FUNCTION_BLOCK fbSliderWithGripperEM EXTENDS fbEM
VAR
	i : INT;
	state : INT;
	initial: BOOL := TRUE;
	servo_GO: BOOL;
	
	fbSignalSim: fbSignalSimSliderWithGripper;
END_VAR
VAR_INPUT
	
END_VAR
VAR_OUTPUT
	
END_VAR

(*
THIS fb use IOs listed below
DATA.I[1] -> true when gripper closed
DATA.I[2] -> true when gripper opened
DATA.I[3] -> part present
DATA.Q[1] -> 1 CLOSE / 0 OPEN gripper
DATA.Q[3] -> SERVO_GO
DATA.pick_pos -> desired pick position
DATA.drop_pos -> desired drop position
DATA.act_pos -> actual postition ( resolved in SIM or SERVO_HANDLER)
DATA.give_pos -> moves desired position into SIM or SERVO_HANDLER)
*)

GetUnCmd();
fbSignalSim(
	em := em,
	EnableSim := EnableSim,
	CmdSim := CmdSim
);

IF initial THEN // AFTER START OF PLC ENTER Undefined state
	state:=0;
	//em.CMD := E_CMD.powerOn; //// MAKES SENSE? <- no it doesnt because you change input 
	initial:= FALSE;
	 em.Config.Data.pick_pos:=10; 
	 em.Config.Data.pick_pos:=200;
	
END_IF

IF em.CMD = E_CMD.abort THEN
	state:=65;
END_IF

IF em.CMD = E_CMD.stop THEN
	state:=70;
END_IF

CASE state OF
	
	0:		//RESETTING
		em.Status := E_Status.resetting;	
		
		
		IF  em.Config.Data.pick_pos = em.Config.Data.act_pos THEN   // ACTUAL POS READ FROM SERVO HANDLER / FOR NOW FROM SIGNAL SIM
				
				servo_GO:=FALSE;
				state :=30; // IF gripper at PICK_pos go to idle
		END_IF
		IF em.CMD = E_CMD.reset THEN 		
				em.Config.Data.give_pos:=em.Config.Data.pick_pos;
				servo_GO:=TRUE;
				
				//// IF gripper pos unknown move to PICK
				//SERVO_HANDLER HAS TO KNOW THE CASE STEP TO DECIDE WHERE TO MOVE 			 
				//HERE SIGNAL SIM HANDLE THIS		
		END_IF
		

	
	30:		//IDLE
		em.Status := E_Status.idle;
		IF em.CMD = E_CMD.start THEN 
			state :=40;
		END_IF
		

	40:		//EXECUTE.1
		em.Status := E_Status.execute;
				
		//Close gripper when part present
		IF em.Config.Data.I[3]  THEN 
			em.Config.Data.Q[1]:= TRUE; //CLOSE GRIPPER
		END_IF
		
		//When Gripper closed --> state 41
		IF em.Config.Data.I[1] = TRUE AND em.Config.Data.I[2]=FALSE THEN
			state:=41;
		END_IF

	41:		//EXECUTE.2 ORDER TO MOVE TO CHOOSEN POSITION
		em.Status := E_Status.execute;
		em.Config.Data.give_pos := em.Config.Data.drop_pos;
		servo_GO:=TRUE; 							
		IF em.Config.Data.act_pos = em.Config.Data.drop_pos THEN
		servo_GO:=FALSE;
		state:=42;										
		END_IF


	42:		//EXECUTE.3 OPEN GRIPPER
	
		em.Status := E_Status.execute;
		em.Config.Data.Q[1]:=FALSE; //OPEN GRIPPER
		IF em.Config.Data.I[1] = FALSE AND em.Config.Data.I[2]=TRUE THEN
			state:=43;
		END_IF
		
			
	43:		//EXECUTE.4 MOVING PICK_POS WITHOUT PART

		em.Status := E_Status.execute;
		IF NOT em.Config.Data.I[3]  
			AND em.Config.Data.act_pos =em.Config.Data.drop_pos THEN//when part gone
			em.Config.Data.give_pos:=em.Config.Data.pick_pos;
			servo_GO:=TRUE;//GO 
			//SERVO_HANDLER HAS TO KNOW THE CASE STEP TO DECIDE WHERE TO MOVE 			 
			//HERE SIGNAL SIM HANDLE THIS	
		END_IF
		
		IF em.Config.Data.act_pos = em.Config.Data.pick_pos THEN
			servo_GO:=FALSE;
			state:=40;
			//em.Config.Data.pick_pos:= -1;
			//em.Config.Data.drop_pos:= -1;
		END_IF
	
	
	65:		//ABORTED

		em.Status := E_Status.aborted;	
		servo_GO:=FALSE;
		IF em.CMD = E_CMD.clear THEN
			state := 70;
		END_IF;


	70: //STOPPED

		em.Status := E_Status.stopped;	
		servo_GO:=FALSE;
		IF em.CMD = E_CMD.reset THEN
			state:=0;
		END_IF

	
END_CASE



em.SequenceStep:=state;       //pass sequence step outside to SimSignal

em.Config.Data.Q[3]:=servo_GO;//Q[3] alias





(*  SERVO HANDLER LOGIC
	IF SERVO_GO AND STATE = 0 THEN MOVE_TO_PICK_POS
	IF SERVO_GO AND STATE = 41 THEN MOVE_TO_DROP_POS
	IF SERVO_GO AND STATE = 44 THEN MOVE_TO_PICK_POS  *)

(*BEST MOMENT TO WRITE DESIRED pick_pos or drop_pos is STATE 30 or 40*)

END_FUNCTION_BLOCK

(* stored: Version 1.1.0.1, ProductVersion 3.1.4024.12
   POU fbSliderWithGripperEM: Id {262a0099-d26a-4a20-85d1-5e68be47c9f0}, SpecialFunc None *)
